(* Schneider Machine Expert - Basic project Timer Project = 4, file version 2.7.0.0 *)
(* ProjectInformations: Name=New project *)

HARDWARE
  Cpu 0: TM221M16R/G
  EthernetConfiguration: NetworkName=M221, IpAllocationMode=FixedAddress, IpAddress=0.0.0.0, SubnetMask=0.0.0.0
  SerialLineConfiguration: Baud=Baud19200, Parity=ParityEven, DataBits=DataBits8, StopBits=StopBits1, PhysicalMedium=PhysicalMediumRs485, TransmissionMode=TransmissionModeModbusRtu, SlaveId=1, Addressing=SlaveAddressing
  MastTask: UsePeriodScanMode=false, PeriodScan=100
  FastTask: Period=255
  CpuBehavior: StartingMode=StartAsPreviousState, AutoSaveRamOnEeprom=true, WatchdogPeriod=250

SYMBOLS  (address, symbol, comment, settings)
  %TM0        [Type=TOF, Preset=5, Base=OneSecond]
  %TM1        [Preset=5, Base=OneSecond]

POU New POU
  (* SectionNumber=1 *)

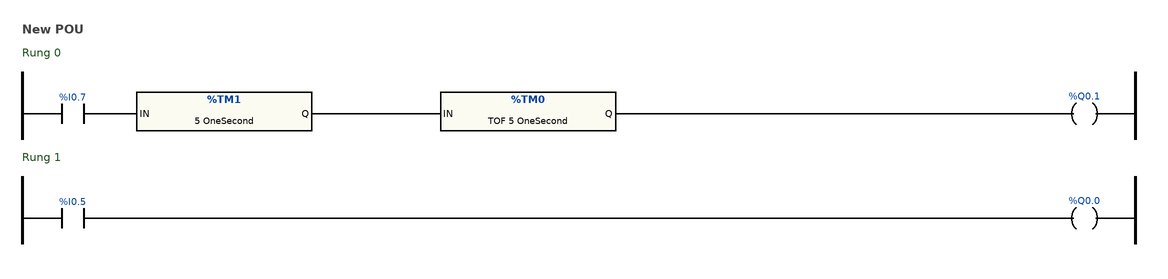

// Rung 0
  LD 1
  MULTIFB
  BLK %TM1
  LD 1
  AND %I0.7
  IN
  OUT_BLK
  LD Q
  ST %MW2009:X0
  END_BLK
  BLK %TM0
  LD %MW2009:X0
  IN
  OUT_BLK
  LD Q
  ST %Q0.1
  END_BLK
  MULTIFB
  // as ST:
  //   %TM1(IN := %I0.7);
  //   %TM0(IN := %TM1.Q);
  //   %Q0.1 := %TM0.Q;

// Rung 1
  LD %I0.5
  ST %Q0.0
  // as ST:
  //   %Q0.0 := %I0.5;
